FUNCTION OSCAT_DW_TO_REAL : REAL
// E. Foy (2021-08-30): Copied from OSCAT library.
VAR_INPUT
	X : DWORD;
END_VAR
VAR
	pt : POINTER TO REAL;
END_VAR

(*
version 1.0	18. apr. 2008
programmer 	hugo
tested by		tobias

this function converts a DWORD to REAL in a bitwise manner.
*)

pt := ADR(X);
OSCAT_DW_TO_REAL := pt^;

(* revision history
hm	18. apr. 2008
	original version

*)

END_FUNCTION

(* stored: Version 1.1.0.1, ProductVersion 3.1.4024.9
   POU OSCAT_DW_TO_REAL: Id {71677e02-0b54-4fd8-8916-eae6a13cd55c}, SpecialFunc None *)
